// TwinCAT 3 PLC project Untitled1
// Title: Lib
// Company: Terza-Automation
// ProjectVersion: 0.1
// ProgramVersion: 3.1.4024.0
// libraries:
//   Tc2_ModbusRTU, * (Beckhoff Automation GmbH)
//   Tc2_Standard, * (Beckhoff Automation GmbH)
//   Tc2_System, * (Beckhoff Automation GmbH)
//   Tc2_Utilities, * (Beckhoff Automation GmbH)
//   Tc3_Module, * (Beckhoff Automation GmbH)
// project tree:
//   DUTs/ Beckhoff_AI.TcDUT, ModbusRealWordUnion.TcDUT, RTU_EM.TcDUT, RTU_STS.TcDUT, RTU_THT.TcDUT
//   / GlobalTextList.TcGTLO, PlcTask.TcTTO
//   GVLs/ GVL.TcGVL, GVL_DataHalls.TcGVL, GVL_DECI.TcGVL, GVL_Electrical.TcGVL, GVL_EM.TcGVL, GVL_STS.TcGVL, GVL_THT.TcGVL
//   POUs/ AccumDDHHMM.TcPOU, AccumTimes.TcPOU, CAC_Analog.TcPOU, CAC_Average.TcPOU, CAC_Mirror.TcPOU, MAIN.TcPOU, ModbusRTU_STS.TcPOU, ModbusRTU_THT.TcPOU, Modbus_EM.TcPOU, OneATS.TcPOU, OneCRAH.TcPOU, OneDI.TcPOU, OneEnergyMeter.TcPOU, OneFire_Suppr.TcPOU, OneGen.TcPOU, OneIDF.TcPOU, OneMYAUX_GLP.TcPOU, OnePDU.TcPOU, OneSTS.TcPOU, OneSWBL.TcPOU, OneTie_BRK.TcPOU, OneUPS.TcPOU
//   Version/ Global_Version.TcGVL
// real-time tasks:
//   TASK PlcTask: cycle T#10ms, priority 20, ADS port 350

CONFIGURATION Untitled1
    RESOURCE PLC ON TwinCAT3
        TASK PlcTask(INTERVAL := T#10ms, PRIORITY := 20);
        PROGRAM MAIN WITH PlcTask : MAIN;
    END_RESOURCE
END_CONFIGURATION

// ---- DUTs/Beckhoff_AI.TcDUT
TYPE Beckhoff_AI :
STRUCT
	rawValue : WORD;
	OutOfRange : BOOL;
	Offline : BOOL;
	Value : REAL;
	
END_STRUCT
END_TYPE

// ---- DUTs/ModbusRealWordUnion.TcDUT
TYPE ModbusRealWordUnion :
UNION
	realValue : REAL;
	wordValue : ARRAY[1..2] OF WORD;
END_UNION
END_TYPE

// ---- DUTs/RTU_EM.TcDUT
TYPE RTU_EM :
STRUCT
	Status : WORD;
	Operating_Hrs : REAL;
	Energy : REAL;
	Volume : REAL;
	Supply_Temp : REAL;
	Return_Temp : REAL;
	Temp_Diff : REAL;
	CommsError : BOOL;
	CommsErrorCode : INT;
END_STRUCT
END_TYPE

// ---- DUTs/RTU_STS.TcDUT
TYPE RTU_STS :
STRUCT
	CommsError : BOOL;
	CommsErrorCode : INT;

	PRI_VA : REAL;
	PRI_VB : REAL;
	PRI_VC : REAL;
	OTP_VA : REAL;
	OTP_VB : REAL;
	OTP_VC : REAL;
	AMPSA : REAL;
	AMPSB : REAL;
	AMPSC : REAL;
	FREQ : REAL;
	SEC_VA : REAL;
	SEC_VB : REAL;
	SEC_VC : REAL;
	OTP_LOAD_A : REAL;
	OTP_LOAD_B : REAL;
	OTP_LOAD_C : REAL;
	COM_ALM : BOOL;
	OTP_KW_A : REAL;
	OTP_KW_B : REAL;
	OTP_KW_C : REAL;
	OTP_KVA_A : REAL;
	OTP_KVA_B : REAL;
	OTP_KVA_C : REAL;
	PF_A : REAL;
	PF_B : REAL;
	PF_C : REAL;

	OTP_BKR_OPN : BOOL;
	L1_INP_BKR_OPN : BOOL;
	L2_INP_BKR_OPN : BOOL;
	L1_BYP_BKR_TRP : BOOL;
	L2_BYP_BKR_TRP : BOOL;
	OTP_BKR_TRP : BOOL;
	L1_INP_BKR_TRP : BOOL;
	L2_INP_BKR_TRP : BOOL;
	FANS_FAIL : BOOL;
	
END_STRUCT
END_TYPE

// ---- DUTs/RTU_THT.TcDUT
TYPE RTU_THT :
STRUCT
	Temp : REAL;
	RH : REAL;
	Temp_OOR : BOOL;
	RH_OOR : BOOL;
	CommsError : BOOL;
	CommsErrorCode : INT;
END_STRUCT
END_TYPE

// ---- GVLs/GVL.TcGVL
	{attribute 'qualified_only'}
VAR_GLOBAL
	mb_Input_Coils    	:	ARRAY [0..511] OF BOOL;
	mb_Output_Coils 	:   ARRAY [0..511] OF BOOL;
 	mb_Input_Registers 	:   ARRAY [0..511] OF WORD;
 	mb_Output_Registers :   ARRAY [0..255] OF WORD;
	
	nInputCoilIndex: INT;
	nOutputCoilIndex: INT;
	nInputRegisterIndex: INT;
	nOutputRegisterIndex: INT;
END_VAR

// ---- GVLs/GVL_DataHalls.TcGVL
{attribute 'qualified_only'}

VAR_GLOBAL CONSTANT
	StartInputCoilIndex_CRAH : INT := 0;			// uses 0-95
	StartInputCoilIndex_PDU : INT := 96;			// uses 96-239
	StartInputCoilIndex_CAC : INT := 0;				// not used
	StartInputCoilIndex_OtherDIs : INT := 275;		// uses 275-294
	StartInputCoilIndex_E_METER : INT := 295;		// uses 295-296
	StartInputCoilIndex_IO : INT := 297;			// uses 297-336
	StartInputCoilIndex_IDF : INT := 240;           // uses 240-257
	StartInputCoilIndex_GLP : INT := 258;           // uses 258-266
	StartInputCoilIndex_ATS : INT := 267;           // uses 267-274
    
	StartOutputCoilIndex_CRAH : INT := 0;			// uses 0-31
	StartOutputCoilIndex_PDU : INT := 0;			// not used
	StartOutputCoilIndex_CAC : INT := 35;			// uses 35-402
	StartOutputCoilIndex_OtherDIs : INT := 0;		// not used
	StartoutputCoilIndex_E_METER : INT := 0;		// not used
	StartoutputCoilIndex_IO : INT := 0;				// not used
	StartoutputCoilIndex_IDF : INT := 0;	        // not used
	StartoutputCoilIndex_GLP : INT := 0;	        // not used
	StartoutputCoilIndex_ATS : INT := 32;	        // uses 32-34
	
	StartInputRegisterIndex_CRAH: INT := 0;			// uses 0-127
	StartInputRegisterIndex_PDU: INT := 0;			// not used
	StartInputRegisterIndex_CAC: INT := 0;			// not used
	StartInputRegisterIndex_OtherDIs : INT := 0;	// not used
	StartInputRegisterIndex_E_METER : INT := 128;	// uses 128-254
    StartInputRegisterIndex_IO : INT := 0;			// not used
	StartInputRegisterIndex_IDF : INT := 0;			// not used
	StartInputRegisterIndex_GLP : INT := 0;			// not used
	StartInputRegisterIndex_ATS : INT := 0;			// not used
		
	StartOutputRegisterIndex_CRAH: INT := 0;		// not used
	StartOutputRegisterIndex_PDU: INT := 0;			// not used
	StartOutputRegisterIndex_CAC: INT := 0;			// uses 0-143
	StartOutputRegisterIndex_OtherDIs : INT := 0;	// not used
	StartoutputRegisterIndex_E_METER : INT := 0;	// not used
	StartoutputRegisterIndex_IO : INT := 0;			// not used
	StartoutputRegisterIndex_IDF : INT := 0;		// not used
	StartoutputRegisterIndex_GLP : INT := 0;		// not used
	StartoutputRegisterIndex_ATS : INT := 0;		// not used
	
END_VAR

// ---- GVLs/GVL_DECI.TcGVL
{attribute 'qualified_only'}
VAR_GLOBAL
	//Date and Time
    fbGetLocalSystemTime: FB_LocalSystemTime;
	sSystemDateTime : STRING;
	sSystemTime : STRING;
	sSystemDate : STRING;	

	// Coupler state - a UINT that should be 8 if its healthy
	CouplerStatus AT %I* : UINT;
	Term02Status AT %I* : WORD;
	Term03Status AT %I* : WORD;
	Term04Status AT %I* : WORD;
	Term05Status AT %I* : WORD;
	Term06Status AT %I* : WORD;
	Term07Status AT %I* : WORD;
	Term08Status AT %I* : WORD;
	Term09Status AT %I* : WORD;
	Term10Status AT %I* : WORD;
	Term11Status AT %I* : WORD;
	Term12Status AT %I* : WORD;
	Term13Status AT %I* : WORD;
	Term14Status AT %I* : WORD;
	Term15Status AT %I* : WORD;
	Term16Status AT %I* : WORD;
	Term17Status AT %I* : WORD;
	Term18Status AT %I* : WORD;
	Term19Status AT %I* : WORD;
	Term20Status AT %I* : WORD;
	Term21Status AT %I* : WORD;
	Term22Status AT %I* : WORD;
	Term23Status AT %I* : WORD;
	Term24Status AT %I* : WORD;
	Term25Status AT %I* : WORD;
	Term26Status AT %I* : WORD;
	Term27Status AT %I* : WORD;
	Term28Status AT %I* : WORD;
	Term29Status AT %I* : WORD;
	Term30Status AT %I* : WORD;
	Term31Status AT %I* : WORD;
	Term32Status AT %I* : WORD;
	Term33Status AT %I* : WORD;
	Term34Status AT %I* : WORD;
	Term35Status AT %I* : WORD;
	Term36Status AT %I* : WORD;
    Term37Status AT %I* : WORD;
	
	// I/O module status
	CouplerOffline : BOOL;
	Term02Offline : BOOL;
	Term03Offline : BOOL;
	Term04Offline : BOOL;
	Term05Offline : BOOL;
	Term06Offline : BOOL;
	Term07Offline : BOOL;
	Term08Offline : BOOL;
	Term09Offline : BOOL;
	Term10Offline : BOOL;
	Term11Offline : BOOL;
	Term12Offline : BOOL;
	Term13Offline : BOOL;
	Term14Offline : BOOL;
	Term15Offline : BOOL;
	Term16Offline : BOOL;
	Term17Offline : BOOL;
	Term18Offline : BOOL;
	Term19Offline : BOOL;
	Term20Offline : BOOL;
	Term21Offline : BOOL;
	Term22Offline : BOOL;
	Term23Offline : BOOL;
	Term24Offline : BOOL;
	Term25Offline : BOOL;
	Term26Offline : BOOL;
	Term27Offline : BOOL;
	Term28Offline : BOOL;
	Term29Offline : BOOL;
	Term30Offline : BOOL;
	Term31Offline : BOOL;
	Term32Offline : BOOL;
	Term33Offline : BOOL;
	Term34Offline : BOOL;
	Term35Offline : BOOL;
	Term36Offline : BOOL;
	Term37Offline : BOOL;
	
END_VAR

VAR_GLOBAL CONSTANT
	

END_VAR

// ---- GVLs/GVL_Electrical.TcGVL
{attribute 'qualified_only'}


VAR_GLOBAL CONSTANT
	StartInputCoilIndex_CRAH : INT := 0;			     // uses 0-29
	StartInputCoilIndex_SWBL : INT := 30;			     // uses 30-89
	StartInputCoilIndex_CAC : INT := 0;				     // not used
	StartInputCoilIndex_OtherDIs : INT := 297;		     // uses 297-330
	StartInputCoilIndex_TX : INT := 227;			     // uses 227-234
	StartInputCoilIndex_GEN : INT := 235;			     // uses 235-244
	StartInputCoilIndex_UPS : INT := 245;			     // uses 245-260
	StartInputCoilIndex_EMG_LIT : INT := 261;			 // uses 261-272
	StartInputCoilIndex_Fire_Suppr : INT := 273;		 // uses 273-296
	StartInputCoilIndex_ATS : INT := 219;                // uses 219-226
	StartInputCoilIndex_MYAUX_GLP : INT := 210;          // uses 210-218
	StartInputCoilIndex_Tie_BRK : INT := 90;             // uses 90-97
	StartInputCoilIndex_STS : INT := 98;			     // uses 98-209
	StartInputCoilIndex_STSRTU : INT := 331;		     // uses 331-407
 	StartInputCoilIndex_IO : INT := 408;				 // uses 408-430
 	StartInputCoilIndex_RTUStat : INT := 431;		 	 // uses 431-440
   
	StartOutputCoilIndex_CRAH : INT := 0;			     // uses 0-11
	StartOutputCoilIndex_SWBL : INT := 0;			     // not used
	StartOutputCoilIndex_CAC : INT := 23;			     // uses 23-52
	StartOutputCoilIndex_OtherDIs : INT := 0;		     // not used 
	StartOutputCoilIndex_TX : INT := 0;				     // not used
	StartOutputCoilIndex_GEN : INT := 53;	             // uses 53-54
	StartOutputCoilIndex_UPS : INT := 0;	             // not used
	StartOutputCoilIndex_EMG_LIT : INT := 0;	         // not used 
	StartOutputCoilIndex_Fire_Suppr : INT := 0;	         // not used
	StartOutputCoilIndex_ATS : INT := 20;	             // uses 20-22
	StartOutputCoilIndex_MYAUX_GLP : INT := 0;	         // not used
	StartOutputCoilIndex_Tie_BRK : INT := 0;	         // not used
	StartOutputCoilIndex_STS : INT := 12;	             // uses 12-19
	StartOutputCoilIndex_STSRTU : INT := 0;	             // not used
 	StartOutputCoilIndex_IO : INT := 0;				 	 // not used
 	StartOutputCoilIndex_RTUStat : INT := 0;			 // not used
	
	StartInputRegisterIndex_CRAH: INT := 0;			     // uses 0-46
	StartInputRegisterIndex_SWBL: INT := 0;			     // not used
	StartInputRegisterIndex_CAC: INT := 0;			     // not used
	StartInputRegisterIndex_OtherDIs : INT := 0;	     // not used
    StartInputRegisterIndex_TX : INT := 0;			     // not used
	StartInputRegisterIndex_GEN : INT := 0;			     // not used
	StartInputRegisterIndex_UPS : INT := 0;			     // not used
	StartInputRegisterIndex_EMG_LIT : INT := 0;			 // not used
	StartInputRegisterIndex_Fire_Suppr : INT := 0;	     // not used
	StartInputRegisterIndex_ATS : INT := 0;			     // not used
	StartInputRegisterIndex_MYAUX_GLP : INT := 0;	     // not used
	StartInputRegisterIndex_Tie_BRK : INT := 0;	         // not used
	StartInputRegisterIndex_STS : INT := 0;			     // not used
	StartInputRegisterIndex_STSRTU : INT := 61;			 // uses 61-460
 	StartInputRegisterIndex_IO : INT := 0;				 // not used
 	StartInputRegisterIndex_RTUStat : INT := 47;		 // uses 47-56
		
	StartOutputRegisterIndex_CRAH: INT := 0;		     // not used
	StartOutputRegisterIndex_SWBL: INT := 0;		     // not used
	StartOutputRegisterIndex_CAC: INT := 0;			     // uses 0-10
	StartOutputRegisterIndex_OtherDIs : INT := 0;	     // not used
	StartOutputRegisterIndex_TX : INT := 0;			     // not used
	StartOutputRegisterIndex_GEN : INT := 0;			 // not used
	StartOutputRegisterIndex_UPS : INT := 0;			 // not used
	StartOutputRegisterIndex_EMG_LIT : INT := 0;	     // not used
	StartOutputRegisterIndex_Fire_Suppr : INT := 0;	     // not used
	StartOutputRegisterIndex_ATS : INT := 0;		     // not used
	StartOutputRegisterIndex_MYAUX_GLP : INT := 0;		 // not used
	StartOutputRegisterIndex_Tie_BRK : INT := 0;		 // not used
	StartOutputRegisterIndex_STS : INT := 0;			 // not used
	StartOutputRegisterIndex_STSRTU : INT := 0;			 // not used
 	StartOutputRegisterIndex_IO : INT := 0;				 // not used
 	StartOutputRegisterIndex_RTUStat : INT := 0;		 // not used
	
END_VAR

// ---- GVLs/GVL_EM.TcGVL
{attribute 'qualified_only'}
VAR_GLOBAL
	EM : ARRAY [1..2] OF RTU_EM;
END_VAR

// ---- GVLs/GVL_STS.TcGVL
{attribute 'qualified_only'}
VAR_GLOBAL
	STS : ARRAY [1..10] OF RTU_STS;
END_VAR

// ---- GVLs/GVL_THT.TcGVL
{attribute 'qualified_only'}
VAR_GLOBAL
	THT : ARRAY [1..14] OF RTU_THT;
END_VAR


VAR_GLOBAL CONSTANT
	Temp_OOR_Min : REAL :=   0.0;
	Temp_OOR_Max : REAL :=  50.0;
	RH_OOR_Min   : REAL :=   0.0;
	RH_OOR_Max   : REAL := 100.0;
END_VAR

// ---- Version/Global_Version.TcGVL
{attribute 'TcGenerated'}
{attribute 'no-analysis'}
{attribute 'linkalways'}
// This function has been automatically generated from the project information.
VAR_GLOBAL CONSTANT
	{attribute 'const_non_replaced'}
	stLibVersion_Lib : ST_LibVersion := (iMajor := 0, iMinor := 1, iBuild := 0, iRevision := 0, nFlags := 0, sVersion := '0.1');
END_VAR

// ---- POUs/MAIN.TcPOU
PROGRAM MAIN
VAR
	foo:AccumDDHHMM;
	in1 AT %I* : BOOL;
	
	foo1: BOOL;
	foo2: BOOL;
	foo3: BOOL;
	
	foo4:STRING;
	
END_VAR

foo(State:=foo1 , Retentive:= foo2, Reset:=foo3);

foo4:=foo.DispayTime;

END_PROGRAM

// ---- POUs/AccumDDHHMM.TcPOU
FUNCTION_BLOCK AccumDDHHMM
VAR_INPUT
	State:BOOL;
	Retentive:BOOL;
	Reset:BOOL;
END_VAR

VAR PERSISTENT
	Mins:WORD;
	Hrs:WORD;
	Sec:WORD;
	Days:WORD;
END_VAR

VAR
	DispayTime:STRING;
	timer:TON;
	timerPT:TIME:=T#1M;
	StateToOff: F_TRIG;
    
END_VAR

VAR_TEMP
	displayTimeFormat: FB_FormatString;	
	foo:DINT;
END_VAR
VAR // added by the converter: edge detectors and wires of the graphical bodies
    _w1, _w2, _w3 : BOOL;
END_VAR

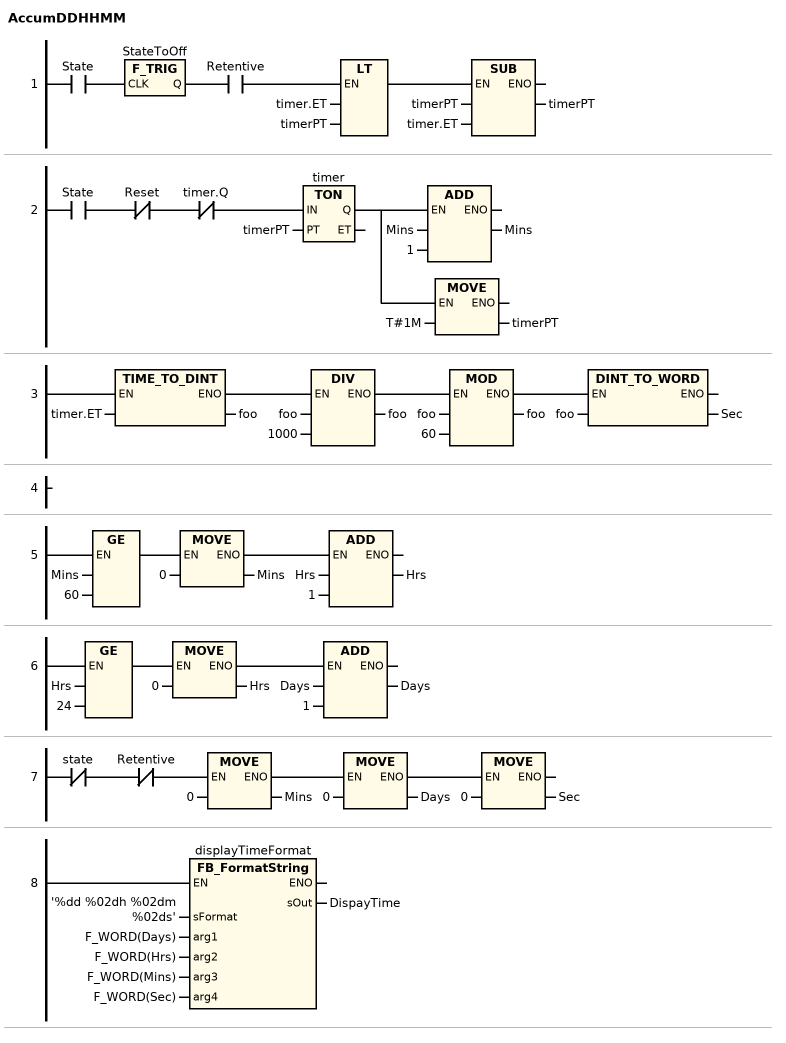
// NETWORK 1
StateToOff(CLK := State); // F_TRIG
IF StateToOff.Q AND Retentive AND timer.ET < timerPT THEN timerPT := timerPT - timer.ET; END_IF

// NETWORK 2
timer(IN := State AND NOT Reset AND NOT timer.Q, PT := timerPT); // TON
IF timer.Q THEN Mins := Mins + 1; END_IF
IF timer.Q THEN timerPT := T#1M; END_IF

// NETWORK 3
foo := TIME_TO_DINT(timer.ET);
foo := foo / 1000;
foo := foo MOD 60;
Sec := DINT_TO_WORD(foo);

// NETWORK 4

// NETWORK 5
_w1 := Mins >= 60;
IF _w1 THEN Mins := 0; END_IF
IF _w1 THEN Hrs := Hrs + 1; END_IF

// NETWORK 6
_w2 := Hrs >= 24;
IF _w2 THEN Hrs := 0; END_IF
IF _w2 THEN Days := Days + 1; END_IF

// NETWORK 7
_w3 := NOT state AND NOT Retentive;
IF _w3 THEN Mins := 0; END_IF
IF _w3 THEN Days := 0; END_IF
IF _w3 THEN Sec := 0; END_IF

// NETWORK 8
displayTimeFormat(
    sFormat := '%dd %02dh %02dm %02ds',
    arg1 := F_WORD(Days),
    arg2 := F_WORD(Hrs),
    arg3 := F_WORD(Mins),
    arg4 := F_WORD(Sec),
    sOut => DispayTime); // FB_FormatString

END_FUNCTION_BLOCK

// ---- POUs/AccumTimes.TcPOU
FUNCTION_BLOCK AccumTimes
VAR_INPUT
	State:BOOL;
END_VAR
VAR PERSISTENT
	Num:WORD;
	ResetAccum:BOOL;
	
	cntOn:CTU;
	Accum:AccumDDHHMM;
	On:AccumDDHHMM;
	Off:AccumDDHHMM;
END_VAR

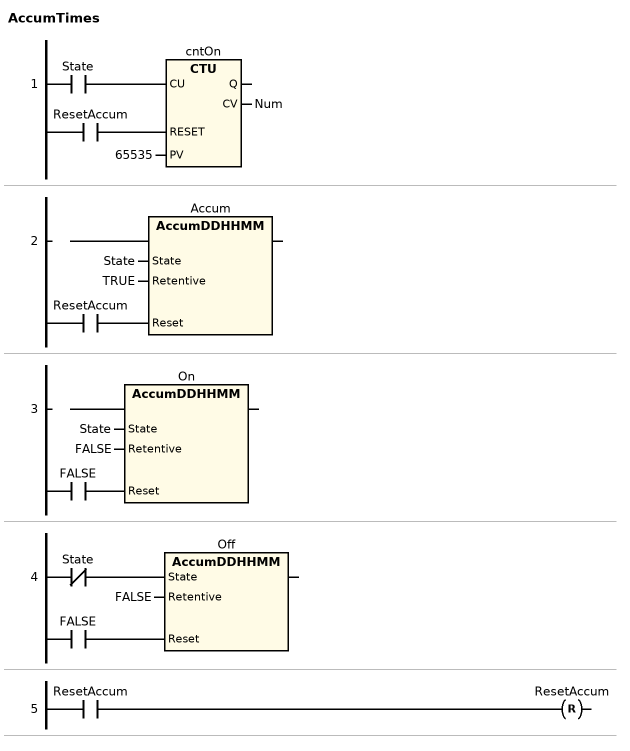
// NETWORK 1
cntOn(CU := State, RESET := ResetAccum, PV := 65535, CV => Num); // CTU

// NETWORK 2
Accum(State := State, Retentive := TRUE, Reset := ResetAccum); // AccumDDHHMM

// NETWORK 3
On(State := State, Retentive := FALSE, Reset := FALSE); // AccumDDHHMM

// NETWORK 4
Off(State := NOT State, Retentive := FALSE, Reset := FALSE); // AccumDDHHMM

// NETWORK 5
ResetAccum R= ResetAccum;

END_FUNCTION_BLOCK

// ---- POUs/CAC_Analog.TcPOU
FUNCTION_BLOCK CAC_Analog
VAR_INPUT
	Value : REAL;			// from EtherCAT I/O
	OutOfRange : BOOL;		// from EtherCAT I/O
	Offline: BOOL;			// from EtherCAT I/O
END_VAR

VAR
	SetInclude : BOOL;		// set on graphics, reset by WinCC OA
	SetExclude : BOOL;		// set on graphics, reset by WinCC OA
	Excluded : BOOL;		// maintained by WinCC OA
	Alarm : BOOL;			// maintained by WinCC OA
	SetIncludeTrig: R_TRIG;	
	SetExcludeTrig: R_TRIG;
END_VAR
VAR_TEMP
	i: INT;	
	modbusReal : ModbusRealWordUnion;
END_VAR


i := GVL.nOutputRegisterIndex;
modbusReal.realValue :=Value;
GVL.mb_Output_Registers[i+0]:= modbusReal.wordValue[1];
GVL.mb_Output_Registers[i+1]:= modbusReal.wordValue[2];

i := GVL.nOutputCoilIndex;
GVL.mb_Output_Coils[i+0]:=OutOfRange;
GVL.mb_Output_Coils[i+1]:=Offline;

SetIncludeTRig(CLK:=SetInclude);

IF SetIncludeTRig.Q THEN
	GVL.mb_Output_Coils[i+2]:=TRUE;
ELSIF SetInclude AND GVL.mb_Output_Coils[i+2] =0 THEN 
	SetInclude:= FALSE;
END_IF

END_FUNCTION_BLOCK

// ---- POUs/CAC_Average.TcPOU
FUNCTION_BLOCK CAC_Average
VAR_INPUT
END_VAR
VAR_OUTPUT
END_VAR
VAR
	Value:REAL;
	Alarm: BOOL;
	OutOfRange: BOOL;
	Offline: BOOL;
	
END_VAR

VAR_TEMP
	i : INT;
	modbusReal : ModbusRealWordUnion;
END_VAR


i:=GVL.nOutputRegisterIndex;
modbusReal.wordValue[0]:=GVL.mb_Output_Registers[i+0];
modbusReal.wordValue[1]:=GVL.mb_Output_Registers[i+1];
Value:= modbusReal.realValue;
GVL.nOutputRegisterIndex:=i+2;

i:=GVL.nOutputCoilIndex;
OutOfRange:=FALSE;
Offline:=GVL.mb_Output_Coils[i+0];
Alarm:=GVL.mb_Output_Coils[i+1];
GVL.nOutputCoilIndex:=i+2;

END_FUNCTION_BLOCK

// ---- POUs/CAC_Mirror.TcPOU
FUNCTION_BLOCK CAC_Mirror
VAR_INPUT
END_VAR
VAR_OUTPUT
END_VAR
VAR
	Value : REAL;			// from partner's EtherCAT I/O, via WinCC OA
	OutOfRange : BOOL;		// from partner's EtherCAT I/O, via WinCC OA
	Offline: BOOL;			// from partner's EtherCAT I/O, via WinCC OA
	SetInclude : BOOL;		// set on graphics, reset by WinCC OA
	SetExclude : BOOL;		// set on graphics, reset by WinCC OA
	Excluded : BOOL;		// maintained by WinCC OA
	Alarm : BOOL;			// maintained by WinCC OA
	SetIncludeTrig: R_TRIG;	
	SetExcludeTrig: R_TRIG;
END_VAR

VAR_TEMP
	i: INT;	
	modbusReal : ModbusRealWordUnion;
END_VAR


i := GVL.nOutputRegisterIndex;
modbusReal.wordValue[1] := GVL.mb_Output_Registers[i+0];
modbusReal.wordValue[2] := GVL.mb_Output_Registers[i+1];
Value := modbusReal.realValue;
GVL.nOutputRegisterIndex := i+2;


i := GVL.nOutputCoilIndex;
OutOfRange := GVL.mb_Output_Coils[i+0];
Offline := GVL.mb_Output_Coils[i+1];

SetIncludeTrig(CLK:=SetInclude);
IF SetIncludeTrig.Q THEN
	GVL.mb_Output_Coils[i+2] := TRUE;
ELSIF SetInclude AND GVL.mb_Output_Coils[i+2] = 0 THEN
	SetInclude := FALSE;
END_IF

SetExcludeTrig(CLK:=SetExclude);
IF SetExcludeTrig.Q THEN
	GVL.mb_Output_Coils[i+3] := TRUE;
ELSIF SetExclude AND GVL.mb_Output_Coils[i+3] = 0 THEN
	SetExclude := FALSE;
END_IF

Excluded := GVL.mb_Output_Coils[i+4];
Alarm := GVL.mb_Output_Coils[i+5];
GVL.nOutputCoilIndex := i+6;

END_FUNCTION_BLOCK

// ---- POUs/ModbusRTU_STS.TcPOU
FUNCTION_BLOCK ModbusRTU_STS
VAR_INPUT
	MB_FirstUnitID: BYTE;
	MB_LastUnitID: BYTE;
END_VAR
VAR_OUTPUT
END_VAR
VAR
	ModbusTerm: ModbusRtuMaster_KL6x22B;
	
	MB_UnitID: BYTE:=0;
	MB_Address : WORD := 0;
	MB_Quantity : WORD := 2;
	MB_ReadData : ARRAY[1..15] OF WORD;
	
	MB_TrigRead : BOOL := FALSE;
	MB_CommState:(TRiGGER, TRIGGERED, WAIT_RESPONSE, SETUP_NEXT_MESSAGE) := TRIGGER;
	tmrDelay:TON;
	Execute: INT;
END_VAR

VAR	
	STSNum: INT;
	MessageNum: INT := 1;
END_VAR


VAR CONSTANT
	MAX_MESSAGE_NUM: INT:=1;
	MODBUS_DELAY: TIME:=T#0MS;
END_VAR

IF (MB_UnitID < MB_FirstUnitID) OR (MB_UnitID>MB_LastUnitID) THEN 
	MB_UnitID:=MB_FirstUnitID;
	STSNum:=1;
	MessageNum:=1;
	MB_Address:=1;
	MB_Quantity:=13;
END_IF


ModbusTerm.ReadRegs(
	UnitID:= MB_UnitID, 
	Quantity:= MB_Quantity, 
	MBAddr:= MB_Address-1, 
	cbLength:= SIZEOF(MB_ReadData), 
	pMemoryAddr:= ADR(MB_ReadData), 
	Execute:= MB_TrigRead, 
	Timeout:= T#100MS, 
	BUSY=> , 
	Error=> , 
	ErrorId=> , 
	cbRead=> );
	
	
CASE MB_CommState OF 
	TRiGGER:
		tmrDelay(IN:=TRUE, PT:=MODBUS_DELAY);
		IF tmrDelay.Q THEN 
			MB_TrigRead:=TRUE;
			MB_CommState:=TRIGGERED;		
		END_IF
		
	TRIGGERED:
			tmrDelay(IN:=FALSE, PT:=MODBUS_DELAY);
			MB_TrigRead:=FALSE;
			MB_CommState:=WAIT_RESPONSE;
			
	WAIT_RESPONSE:
			IF NOT ModbusTerm.BUSY THEN
				GVL_STS.STS[STSNum].CommsError:= ModbusTerm.Error;
				GVL_STS.STS[STSNum].CommsErrorCode:= ModbusTerm.ErrorId;
				
				IF NOT ModbusTerm.Error THEN 
					IF MessageNum = 1 THEN // extracts the values in 13 registers #1-13
						GVL_STS.STS[STSNum].PRI_VA := WORD_TO_REAL(MB_ReadData[1]);
						GVL_STS.STS[STSNum].PRI_VB := WORD_TO_REAL(MB_ReadData[2]);
						GVL_STS.STS[STSNum].PRI_VC := WORD_TO_REAL(MB_ReadData[3]);
						GVL_STS.STS[STSNum].PRI_VA := WORD_TO_REAL(MB_ReadData[4]);
						GVL_STS.STS[STSNum].OTP_VB := WORD_TO_REAL(MB_ReadData[5]);
						GVL_STS.STS[STSNum].OTP_VC := WORD_TO_REAL(MB_ReadData[6]);
						GVL_STS.STS[STSNum].AMPSA  := WORD_TO_REAL(MB_ReadData[7]);
						GVL_STS.STS[STSNum].AMPSB  := WORD_TO_REAL(MB_ReadData[8]);
						GVL_STS.STS[STSNum].AMPSC  := WORD_TO_REAL(MB_ReadData[9]);
						GVL_STS.STS[STSNum].FREQ   := WORD_TO_REAL(MB_ReadData[10]);
						GVL_STS.STS[STSNum].SEC_VA := WORD_TO_REAL(MB_ReadData[11]);
						GVL_STS.STS[STSNum].SEC_VB := WORD_TO_REAL(MB_ReadData[12]);
						GVL_STS.STS[STSNum].SEC_VC := WORD_TO_REAL(MB_ReadData[14]);

					 ELSIF MessageNum = 2 THEN // extracts the values in 3 registers #17-19
						GVL_STS.STS[STSNum].OTP_LOAD_A:=WORD_TO_REAL(MB_ReadData[1]);
						GVL_STS.STS[STSNum].OTP_LOAD_B:=WORD_TO_REAL(MB_ReadData[2]);
						GVL_STS.STS[STSNum].OTP_LOAD_C:=WORD_TO_REAL(MB_ReadData[3]);
						
					ELSIF MessageNum = 3 THEN 					
						// common alarm is bit 15 of register 41
						GVL_STS.STS[STSNum].COM_ALM :=MB_ReadData[1].15;
						// other alarms of interest are in register 43 
						GVL_STS.STS[STSNum].OTP_BKR_OPN    := MB_ReadData[3].0;
						GVL_STS.STS[STSNum].L1_INP_BKR_OPN := MB_ReadData[3].1;
						GVL_STS.STS[STSNum].L2_INP_BKR_OPN := MB_ReadData[3].2;
						GVL_STS.STS[STSNum].L1_BYP_BKR_TRP := MB_ReadData[3].3;
						GVL_STS.STS[STSNum].L2_BYP_BKR_TRP := MB_ReadData[3].4;
						GVL_STS.STS[STSNum].OTP_BKR_TRP    := MB_ReadData[3].5;
						GVL_STS.STS[STSNum].L1_INP_BKR_TRP := MB_ReadData[3].6;
						GVL_STS.STS[STSNum].L2_INP_BKR_TRP := MB_ReadData[3].7;
						GVL_STS.STS[STSNum].FANS_FAIL      := MB_ReadData[3].8;	
					
					ELSIF MessageNum = 4 THEN 
						GVL_STS.STS[STSNum].OTP_KW_A  := WORD_TO_REAL(MB_ReadData[1]) / 10.0;
						GVL_STS.STS[STSNum].OTP_KW_B  := WORD_TO_REAL(MB_ReadData[2]) / 10.0;
						GVL_STS.STS[STSNum].OTP_KW_C  := WORD_TO_REAL(MB_ReadData[3]) / 10.0;
						GVL_STS.STS[STSNum].OTP_KVA_A := WORD_TO_REAL(MB_ReadData[4]) / 10.0;
						GVL_STS.STS[STSNum].OTP_KVA_B := WORD_TO_REAL(MB_ReadData[5]) / 10.0;
						GVL_STS.STS[STSNum].OTP_KVA_C := WORD_TO_REAL(MB_ReadData[6]) / 10.0;
					
					ELSIF MessageNum = 5 THEN 
						GVL_STS.STS[STSNum].PF_A := WORD_TO_REAL(MB_ReadData[1]) / 100.0;
						GVL_STS.STS[STSNum].PF_B := WORD_TO_REAL(MB_ReadData[2]) / 100.0;
						GVL_STS.STS[STSNum].PF_C := WORD_TO_REAL(MB_ReadData[3]) / 100.0;	
			
					END_IF
				END_IF
				 
				MB_CommState:=SETUP_NEXT_MESSAGE;
		  END_IF;	 

	SETUP_NEXT_MESSAGE:
		MessageNum:=MessageNum+1;
		
		IF MessageNum > MAX_MESSAGE_NUM THEN 
			MessageNum:=1;
			MB_UnitID:=MB_UnitID+1;
			STSNum:=STSNum+1;	
		END_IF
		
		IF MessageNum = 1  THEN // extracts the values in 13 registers #1-13
			MB_Address:=1;
			MB_Quantity:=13;
			
		ELSIF MessageNum = 2 THEN  // extracts the values in 3 registers #17-19
			MB_Address:=17;
			MB_Quantity:=3;
			 
		ELSIF MessageNum = 3 THEN  // extracts the alarms - 4 registers #41-44
			MB_Address:=41;
			MB_Quantity:=4;
			
		ELSIF MessageNum = 4 THEN  // extracts the values in 6 registers #56-61
			MB_Address:=56;
			MB_Quantity:=6;
			
		ELSIF MessageNum = 5 THEN  // extracts the values in 3 registers #69-71
			MB_Address:=69;
			MB_Quantity:=3;
			
		END_IF 
		
		MB_CommState:=TRiGGER;	
	
END_CASE

END_FUNCTION_BLOCK

// ---- POUs/ModbusRTU_THT.TcPOU
FUNCTION_BLOCK ModbusRTU_THT
VAR_INPUT
	MB_FirstUnitID:BYTE;
	MB_LastUnitID:BYTE;
END_VAR
VAR_OUTPUT
END_VAR
VAR
	ModbusTerm: ModbusRtuMaster_KL6x22B;
	
	MB_UnitID: BYTE:=0;
	MB_Address: WORD:=25;
	MB_Quantity: WORD:=4;
	MB_ReadData: ARRAY[1..2] OF ModbusRealWordUnion;
	
	MB_TrigRead: BOOL:=FALSE;
	MB_CommState: (TRIGGER, TRIGGERED, WAIT_RESPONSE) := TRIGGER;
	tmrDelay: TON;
	

END_VAR

IF (MB_UnitID < MB_FirstUnitID) OR (MB_UnitID>MB_LastUnitID) THEN 
	MB_UnitID:=MB_FirstUnitID;
END_IF


ModbusTerm(
	UnitID:= MB_UnitID, 
	Quantity:= MB_Quantity, 
	MBAddr:= MB_Address, 
	cbLength:= SIZEOF(MB_ReadData), 
	pMemoryAddr:= ADR(MB_ReadData), 
	Execute:= MB_TrigRead, 
	Timeout:= T#2S, 
	BUSY=> , 
	Error=> , 
	ErrorId=> , 
	cbRead=> );
	
CASE MB_CommState OF 
	TRIGGER: 
		tmrDelay(IN:=TRUE, PT:=T#1S);
		IF tmrDelay.Q THEN 
			MB_TrigRead:=TRUE;
			MB_CommState:=TRIGGERED;
		END_IF
		
	TRIGGERED:
		tmrDelay(IN:=FALSE, PT:=T#1S);
		MB_TrigRead:=FALSE;
		MB_CommState:=WAIT_RESPONSE;
		
	WAIT_RESPONSE:
		IF NOT ModbusTerm.BUSY THEN
			GVL_THT.THT[MB_UnitID].CommsError:=ModbusTerm.Error;
			GVL_THT.THT[MB_UnitID].CommsErrorCode:=ModbusTerm.ErrorId;
			
			IF NOT ModbusTerm.Error THEN
				GVL_THT.THT[MB_UnitID].Temp:=MB_ReadData[1].realValue;
				GVL_THT.THT[MB_UnitID].RH  :=MB_ReadData[2].realValue;
				
				GVL_THT.THT[MB_UnitID].Temp_OOR:= (GVL_THT.THT[MB_UnitID].Temp < GVL_THT.Temp_OOR_Min) OR 
												  (GVL_THT.THT[MB_UnitID].Temp > GVL_THT.Temp_OOR_Max);
												  
				GVL_THT.THT[MB_UnitID].RH_OOR:= (GVL_THT.THT[MB_UnitID].RH < GVL_THT.RH_OOR_Min) OR 
												(GVL_THT.THT[MB_UnitID].RH > GVL_THT.RH_OOR_Max);
			END_IF
			
		MB_UnitID   := MB_UnitID+1;
		MB_CommState:= TRIGGER;
		END_IF
END_CASE

END_FUNCTION_BLOCK

// ---- POUs/Modbus_EM.TcPOU
FUNCTION_BLOCK Modbus_EM
VAR_INPUT
	MB_FirstUnitID: BYTE;
	MB_LastUnitID: BYTE;
END_VAR
VAR_OUTPUT
END_VAR
VAR
	ModbusTerm: ModbusRtuMaster_KL6x22B;
	
	MB_UnitID : BYTE := 0;
	MB_Address : WORD := 0;
	MB_Quantity : WORD := 2;
	MB_ReadData : ModbusRealWordUnion;

	MB_TrigRead : BOOL := FALSE;
	MB_CommState: (TRIGGER, TRIGGERED, WAIT_RESPONSE, SETUP_NEXT_MESSAGE) := TRIGGER;
	tmrDelay: TON;
END_VAR

VAR
	EMNum:INT;
	MessageNum:INT;
END_VAR

IF (MB_UnitID < MB_FirstUnitID) OR (MB_UnitID>MB_LastUnitID) THEN 
	
	MB_UnitID:=MB_FirstUnitID;
	EMNum:=1;
	MessageNum:=1;
	MB_Address:=0;

END_IF

ModbusTerm.ReadRegs(
	UnitID:= MB_UnitID, 
	Quantity:= MB_Quantity, 
	MBAddr:= MB_Address, 
	cbLength:= SIZEOF(MB_ReadData), 
	pMemoryAddr:= ADR(MB_ReadData), 
	Execute:= MB_TrigRead, 
	Timeout:= T#2S, 
	BUSY=> , 
	Error=> , 
	ErrorId=> , 
	cbRead=> );
	
CASE MB_CommState OF
	TRIGGER:
			tmrDelay(in:=TRUE, PT:=T#1S);
			
			IF tmrDelay.Q THEN 
				MB_TrigRead:=TRUE;
				MB_CommState:=TRIGGERED;
			END_IF
			
	TRIGGERED:
			tmrDelay(in:=FALSE, PT:=T#1S);
			MB_TrigRead:=FALSE;			
			MB_CommState:=WAIT_RESPONSE;

	WAIT_RESPONSE:
			
			IF NOT ModbusTerm.BUSY THEN 
				GVl_Em.EM[EMNum].CommsError:=ModbusTerm.Error;
				GVl_Em.EM[EMNum].CommsErrorCode:=ModbusTerm.ErrorId;
				
				IF NOT ModbusTerm.Error THEN
					IF MessageNum=1 THEN 
						GVl_Em.EM[EMNum].Status:= MB_ReadData.wordValue[2];
					ELSIF MessageNum=2 THEN 
						GVl_Em.EM[EMNum].Operating_Hrs:= MB_ReadData.realValue;
					ELSIF MessageNum=3 THEN 
						GVl_Em.EM[EMNum].Energy:= MB_ReadData.realValue;
					ELSIF MessageNum=4 THEN 
						GVl_Em.EM[EMNum].Volume:= MB_ReadData.realValue;
					ELSIF MessageNum=5 THEN
						GVl_Em.EM[EMNum].Supply_Temp:= MB_ReadData.realValue;
					ELSIF MessageNum=6 THEN
						GVl_Em.EM[EMNum].Return_Temp:= MB_ReadData.realValue;
					ELSIF MessageNum =7 THEN
						GVl_Em.EM[EMNum].Temp_Diff:= MB_ReadData.realValue;
					END_IF;	
				END_IF
				
				MB_CommState:=SETUP_NEXT_MESSAGE;
				
			END_IF
				
	SETUP_NEXT_MESSAGE:
			MessageNum:=MessageNum+1;
			
			IF MessageNum> 7 THEN 
				
				MessageNum:=1;
				MB_UnitID:=MB_UnitID+1;
				EMNum:=EMNum+1;
				
			END_IF

			IF MessageNum = 1    THEN
				MB_Address:=0; // read status in word 2
			ELSIF MessageNum = 2 THEN 
				MB_Address:=6; // read operating hours
			ELSIF MessageNum = 3 THEN 
				MB_Address:=100; // read energy
			ELSIF MessageNum = 4 THEN 
				MB_Address:=200; // read volume
			ELSIF MessageNum = 5 THEN 
				MB_Address:=800; // read supply temperature
			ELSIF MessageNum = 6 THEN
				MB_Address:=810; // read return temperature
			ELSIF MessageNum = 7 THEN 
				MB_Address:=820;
			END_IF
			
		MB_CommState :=TRIGGER;

END_CASE

END_FUNCTION_BLOCK

// ---- POUs/OneATS.TcPOU
FUNCTION_BLOCK OneATS
VAR_INPUT
	ATS_Avai: BOOL;
	ATS_Avai_Offline: BOOL;	
	ATS_SP1: BOOL;
	ATS_SP1_Offline:BOOL;
	ATS_SP2 : BOOL;
	ATS_SP2_Offline : BOOL;
	ATS_SP0 : BOOL;
	ATS_SP0_Offline : BOOL;
END_VAR

VAR_OUTPUT
	Net_Priority: BOOL;
	Source_Priority: BOOL;
	Inhibited: BOOL;

END_VAR

VAR_TEMP
	i :INT;
END_VAR


i:=GVL.nInputCoilIndex;

GVL.mb_Input_Coils[i+0] := ATS_Avai;
GVL.mb_Input_Coils[i+1] := ATS_Avai_Offline;

GVL.mb_Input_Coils[i+2] := ATS_SP1;
GVL.mb_Input_Coils[i+3] := ATS_SP1_Offline;

GVL.mb_Input_Coils[i+4] := ATS_SP2;
GVL.mb_Input_Coils[i+5] := ATS_SP2_Offline;

GVL.mb_Input_Coils[i+6] := ATS_SP0;
GVL.mb_Input_Coils[i+7] := ATS_SP0_Offline;

i:=GVL.nOutputCoilIndex;
Net_Priority:= GVL.mb_Output_Coils[i+0];
Source_Priority:= GVL.mb_Output_Coils[i+1];
Inhibited:= GVL.mb_Output_Coils[i+2];

GVL.nOutputCoilIndex:=i+3;

END_FUNCTION_BLOCK

// ---- POUs/OneCRAH.TcPOU
FUNCTION_BLOCK OneCRAH
VAR_INPUT
	Running:BOOL;
	Alarm	:BOOL;
	Iso1_1_Sts:BOOL;
	Iso1_2_Sts:BOOL;
	Offline:BOOL;
END_VAR
VAR_OUTPUT
	Enable:BOOL;
END_VAR

VAR PERSISTENT
	Maintenance:BOOL;
	Inhibited:BOOL;
	HOA:WORD;
	Run: AccumTimes;
	Alm: AccumTimes;
	Ena: AccumTimes;
	
END_VAR

VAR_TEMP
	i:INT;
	modbusReal: ModbusRealWordUnion;
END_VAR

Run(State:=Running);
Alm(State:=Alarm);
Ena(State:=Enable);


i:= GVl.nInputCoilIndex;
GVL.mb_Input_Coils[i+0]:= Running;
GVL.mb_Input_Coils[i+1]:= Alarm;
GVL.mb_Input_Coils[i+2]:= Offline;
GVL.mb_Input_Coils[i+3]:= Iso1_1_Sts;
GVL.mb_Input_Coils[i+4]:= Iso1_2_Sts;

GVl.nInputCoilIndex := i+5;

i:=GVL.nOutputCoilIndex;
Enable:= GVL.mb_Output_Coils[i+0];
Inhibited:= GVL.mb_Output_Coils[i+1];
GVL.nOutputCoilIndex:=i+2;


i:=GVL.nInputRegisterIndex;
GVL.mb_Input_Registers[i+0]:= HOA;
GVL.mb_Input_Registers[i+1]:= Run.num;

modbusReal.realValue:= WORD_TO_REAL(Run.Accum.Days) * 24.0 +
					   WORD_TO_REAL(Run.Accum.Hrs)  * 1.0  +
					   WORD_TO_REAL(Run.Accum.Mins) / 60.0;
					   
GVL.mb_Input_Registers[i+2]:= modbusReal.wordValue[1];
GVL.mb_Input_Registers[i+3]:= modbusReal.wordValue[2];

modbusReal.realValue:= WORD_TO_REAL(Run.On.Days) * 24.0 +
					   WORD_TO_REAL(Run.On.Days) * 1.0 +
					   WORD_TO_REAL(Run.On.Mins) / 60.0;
					   
					   
GVL.mb_Input_Registers[i+4]:= modbusReal.wordValue[1];
GVL.mb_Input_Registers[i+5]:= modbusReal.wordValue[2];					   
					   
					   
modbusReal.realValue:= WORD_TO_REAL(Run.Off.Days) * 24.0 +
					   WORD_TO_REAL(Run.Off.Days) * 1.0 +
					   WORD_TO_REAL(Run.Off.Mins) / 60.0;
					   
					   
GVL.mb_Input_Registers[i+6]:= modbusReal.wordValue[1];
GVL.mb_Input_Registers[i+7]:= modbusReal.wordValue[2];

GVL.nInputRegisterIndex:=i+8;

END_FUNCTION_BLOCK

// ---- POUs/OneDI.TcPOU
FUNCTION_BLOCK OneDI
VAR_INPUT
	
	Value  :BOOL;
	Offline:BOOL;
	
END_VAR

VAR_TEMP
	i: INT;
	
END_VAR


i :=GVL.nInputCoilIndex;

GVL.mb_Input_Coils[i+0]:=Value;
GVL.mb_Input_Coils[i+1]:=Offline;

GVL.nInputCoilIndex:= i+2;

END_FUNCTION_BLOCK

// ---- POUs/OneEnergyMeter.TcPOU
FUNCTION_BLOCK OneEnergyMeter
VAR_INPUT
	Status: WORD;
    Operating_Hrs: REAL;
	Energy : REAL;
    Volume: REAL; 
	Supply_Temp: REAL;
	Return_Temp: REAL;
	Temp_Diff: REAL;
	Offline: BOOL;
END_VAR
VAR_OUTPUT
END_VAR
VAR_TEMP
	i : INT;
	modbusReal : ModbusRealWordUnion;
END_VAR


i := GVL.nInputRegisterIndex;

GVL.mb_Input_Registers[i+0] := Status;

modbusReal.realValue := Operating_Hrs;
GVL.mb_Input_Registers[i+2] := modbusReal.wordValue[1];
GVL.mb_Input_Registers[i+3] := modbusReal.wordValue[2];

modbusReal.realValue := Energy;
GVL.mb_Input_Registers[i+4] := modbusReal.wordValue[1];
GVL.mb_Input_Registers[i+5] := modbusReal.wordValue[2];

modbusReal.realValue := Volume;
GVL.mb_Input_Registers[i+6] := modbusReal.wordValue[1];
GVL.mb_Input_Registers[i+7] := modbusReal.wordValue[2];

modbusReal.realValue := Supply_Temp;
GVL.mb_Input_Registers[i+8] := modbusReal.wordValue[1];
GVL.mb_Input_Registers[i+9] := modbusReal.wordValue[2];

modbusReal.realValue := Return_Temp;
GVL.mb_Input_Registers[i+10] := modbusReal.wordValue[1];
GVL.mb_Input_Registers[i+11] := modbusReal.wordValue[2];

modbusReal.realValue := Temp_Diff;
GVL.mb_Input_Registers[i+12] := modbusReal.wordValue[1];
GVL.mb_Input_Registers[i+13] := modbusReal.wordValue[2];

GVL.nInputRegisterIndex := i + 14;


i := GVL.nInputCoilIndex;

GVL.mb_Input_Coils[i+0] := Offline;

GVL.nInputcoilIndex := i + 1;

END_FUNCTION_BLOCK

// ---- POUs/OneFire_Suppr.TcPOU
FUNCTION_BLOCK OneFire_Suppr
VAR_INPUT
	Pnl_Alm : BOOL;
	Pnl_FLT : BOOL;
	Supp_Act : BOOL;
	Fire_Offline : BOOL;
END_VAR
VAR_OUTPUT
END_VAR
VAR_TEMP
	i : INT;
END_VAR


i := GVL.nInputCoilIndex;

GVL.mb_Input_Coils[i+0] := Pnl_Alm;
GVL.mb_Input_Coils[i+1] := Pnl_FLT;
GVL.mb_Input_Coils[i+2] := Supp_Act;
GVL.mb_Input_Coils[i+3] := Fire_Offline;

GVL.nInputCoilIndex := i + 4;

END_FUNCTION_BLOCK

// ---- POUs/OneGen.TcPOU
FUNCTION_BLOCK OneGen
VAR_INPUT
	 Value : BOOL;
	 Offline : BOOL;
END_VAR
VAR_OUTPUT
	  Gen_Oper_Mode : BOOL;
	  Gen_EMG_Shut : BOOL;
END_VAR
VAR_TEMP
	i: INT;
END_VAR

i := GVL.nInputCoilIndex;

GVL.mb_Input_Coils[i+0] := Value;
GVL.mb_Input_Coils[i+1] := Offline;

GVL.nInputCoilIndex := i + 2;

i := GVL.nOutputCoilIndex;

Gen_Oper_Mode := GVL.mb_Output_Coils[i+0];
Gen_EMG_Shut  := GVL.mb_Output_Coils[i+1];

GVL.nOutputCoilIndex := i+2;

END_FUNCTION_BLOCK

// ---- POUs/OneIDF.TcPOU
FUNCTION_BLOCK OneIDF
VAR_INPUT
	sur_STS :BOOL;
	phs_ALM :BOOL;
	sur_phs_offline :BOOL;
	
	BRK115_POS_STS  :BOOL;
	BRK115_TRIP_ALM :BOOL;
	BRK115_offline: BOOL;
	
    BRK125_POS_STS: BOOL;
	BRK125_TRIP_ALM : BOOL; 
	BRK125_offline: BOOL;
		
END_VAR
VAR_OUTPUT
END_VAR

VAR_TEMP
	
	i:INT;

END_VAR

i := GVL.nInputCoilIndex;

GVL.mb_Input_Coils[i+0]:= sur_STS;
GVL.mb_Input_Coils[i+1]:= phs_ALM; 
GVL.mb_Input_Coils[i+2]:= sur_phs_offline;

GVL.mb_Input_Coils[i+3]:= BRK115_POS_STS; 
GVL.mb_Input_Coils[i+4]:= BRK115_TRIP_ALM; 
GVL.mb_Input_Coils[i+5]:= BRK115_offline; 

GVL.mb_Input_Coils[i+6]:= BRK125_POS_STS; 
GVL.mb_Input_Coils[i+7]:= BRK125_TRIP_ALM; 
GVL.mb_Input_Coils[i+8]:= BRK125_offline;

GVL.nInputCoilIndex:=i+9;

END_FUNCTION_BLOCK

// ---- POUs/OneMYAUX_GLP.TcPOU
FUNCTION_BLOCK OneMYAUX_GLP
VAR_INPUT
	sur_STS : BOOL;
	phs_ALM : BOOL;
	sur_phs_offline : BOOL;
	
    BRK119_POS_STS: BOOL;
	BRK119_TRIP_ALM : BOOL; 
	BRK119_offline: BOOL;
	
    BRK129_POS_STS: BOOL;
	BRK129_TRIP_ALM : BOOL; 
	BRK129_offline: BOOL;
END_VAR
VAR_OUTPUT
END_VAR
VAR_TEMP
	i: INT;
END_VAR


i := GVL.nInputCoilIndex;

GVL.mb_Input_Coils[i+0] := sur_STS;
GVL.mb_Input_Coils[i+1] := phs_ALM;
GVL.mb_Input_Coils[i+2] := sur_phs_offline;

GVL.mb_Input_Coils[i+3] := BRK119_POS_STS;
GVL.mb_Input_Coils[i+4] := BRK119_TRIP_ALM;
GVL.mb_Input_Coils[i+5] := BRK119_offline;

GVL.mb_Input_Coils[i+6] := BRK129_POS_STS;
GVL.mb_Input_Coils[i+7] := BRK129_TRIP_ALM;
GVL.mb_Input_Coils[i+8] := BRK129_offline;

GVL.nInputCoilIndex := i + 9;

END_FUNCTION_BLOCK

// ---- POUs/OnePDU.TcPOU
FUNCTION_BLOCK OnePDU
VAR_INPUT
	sur_STS:BOOL;
	phs_ALM:BOOL;
	sur_phs_offline : BOOL;
	
	tvoc_BRK_STS: BOOL;             // CIRCUIT BREAERS
	tvoc_BRK_ALM: BOOL;            // CIRCUIT BREAERS
	tvoc_BRK_offline: BOOL; 
	
	BRK115_POS_STS: BOOL;
	BRK115_TRIP_ALM : BOOL; 
	BRK115_offline: BOOL;
	
	BRK125_POS_STS: BOOL;
	BRK125_TRIP_ALM : BOOL; 
	BRK125_offline: BOOL;
	
	BRK135_POS_STS: BOOL;
	BRK135_TRIP_ALM : BOOL; 
	BRK135_offline: BOOL;
	
	BRK215_POS_STS: BOOL;
	BRK215_TRIP_ALM : BOOL; 
	BRK215_offline: BOOL;
	
	BRK225_POS_STS: BOOL;
	BRK225_TRIP_ALM : BOOL; 
	BRK225_offline: BOOL;
	
	BRK235_POS_STS: BOOL;
	BRK235_TRIP_ALM : BOOL; 
	BRK235_offline: BOOL;
	
	BRK315_POS_STS: BOOL;
	BRK315_TRIP_ALM : BOOL; 
	BRK315_offline: BOOL;
	
	BRK325_POS_STS: BOOL;
	BRK325_TRIP_ALM : BOOL; 
	BRK325_offline: BOOL;
	
	BRK335_POS_STS: BOOL;
	BRK335_TRIP_ALM : BOOL; 
	BRK335_offline: BOOL;
	
	BRK345_POS_STS: BOOL;
	BRK345_TRIP_ALM : BOOL; 
	BRK345_offline: BOOL;
	
END_VAR

VAR_TEMP
	i: INT;
END_VAR


i := GVL.nInputCoilIndex;
GVL.mb_Input_Coils[i+0] := sur_STS;
GVL.mb_Input_Coils[i+1] := phs_ALM;
GVL.mb_Input_Coils[i+2] := sur_phs_offline;

GVL.mb_Input_Coils[i+3] := tvoc_BRK_STS ;
GVL.mb_Input_Coils[i+4] := tvoc_BRK_ALM ;
GVL.mb_Input_Coils[i+5] := tvoc_BRK_offline;

GVL.mb_Input_Coils[i+6] := BRK115_POS_STS;
GVL.mb_Input_Coils[i+7] := BRK115_TRIP_ALM;
GVL.mb_Input_Coils[i+8] := BRK115_offline;

GVL.mb_Input_Coils[i+9] := BRK125_POS_STS;
GVL.mb_Input_Coils[i+10] := BRK125_TRIP_ALM;
GVL.mb_Input_Coils[i+11] := BRK125_offline;

GVL.mb_Input_Coils[i+12] := BRK135_POS_STS;
GVL.mb_Input_Coils[i+13] := BRK135_TRIP_ALM;
GVL.mb_Input_Coils[i+14] := BRK135_offline;

GVL.mb_Input_Coils[i+15] := BRK215_POS_STS;
GVL.mb_Input_Coils[i+16] := BRK215_TRIP_ALM;
GVL.mb_Input_Coils[i+17] := BRK215_offline;

GVL.mb_Input_Coils[i+18] := BRK225_POS_STS;
GVL.mb_Input_Coils[i+19] := BRK225_TRIP_ALM;
GVL.mb_Input_Coils[i+20] := BRK225_offline;

GVL.mb_Input_Coils[i+21] := BRK235_POS_STS;
GVL.mb_Input_Coils[i+22] := BRK235_TRIP_ALM;
GVL.mb_Input_Coils[i+23] := BRK235_offline;

GVL.mb_Input_Coils[i+24] := BRK315_POS_STS;
GVL.mb_Input_Coils[i+25] := BRK315_TRIP_ALM;
GVL.mb_Input_Coils[i+26] := BRK315_offline;

GVL.mb_Input_Coils[i+27] := BRK325_POS_STS;
GVL.mb_Input_Coils[i+28] := BRK325_TRIP_ALM;
GVL.mb_Input_Coils[i+29] := BRK325_offline;

GVL.mb_Input_Coils[i+30] := BRK335_POS_STS;
GVL.mb_Input_Coils[i+31] := BRK335_TRIP_ALM;
GVL.mb_Input_Coils[i+32] := BRK335_Offline;

GVL.mb_Input_Coils[i+33] := BRK345_POS_STS;
GVL.mb_Input_Coils[i+34] := BRK345_TRIP_ALM;
GVL.mb_Input_Coils[i+35] := BRK345_Offline;

GVL.nInputCoilIndex := i + 36;

END_FUNCTION_BLOCK

// ---- POUs/OneSTS.TcPOU
FUNCTION_BLOCK OneSTS
VAR_INPUT
	
	Trans_Inhibt : BOOL;
	Trans_Inhibt_Offline : BOOL;
    Com_Alm : BOOL;
	Com_Alm_Offline: BOOL;
    Fan_Fail : BOOL;
	Fan_Fail_Offline : BOOL;
	
    Load_Line_1 : BOOL;
	Load_Line_1_Offline : BOOL;
    Load_Line_2 : BOOL;
	Load_Line_2_Offline : BOOL;
	
    Load_Line_1_ByPass : BOOL;
	LL_1_ByPass_offline : BOOL;
    Load_Line_2_ByPass : BOOL;
	LL_2_ByPass_offline : BOOL;
	Load_DisCon : BOOL;
	Load_DisCon_Offline : BOOL;

END_VAR
VAR_OUTPUT
	STS_Inhibited : BOOL;
END_VAR
VAR_TEMP
	i : INT;
END_VAR



i := GVL.nInputCoilIndex;
GVL.mb_Input_Coils[i+0] := Trans_Inhibt;
GVL.mb_Input_Coils[i+1] := Trans_Inhibt_Offline;

GVL.mb_Input_Coils[i+2] := Com_Alm;
GVL.mb_Input_Coils[i+3] := Com_Alm_Offline;

GVL.mb_Input_Coils[i+4] := Fan_Fail;
GVL.mb_Input_Coils[i+5] := Fan_Fail_Offline;

GVL.mb_Input_Coils[i+6] := Load_Line_1;
GVL.mb_Input_Coils[i+7] := Load_Line_1_Offline;

GVL.mb_Input_Coils[i+8] := Load_Line_2;
GVL.mb_Input_Coils[i+9] := Load_Line_2_Offline;

GVL.mb_Input_Coils[i+10] := Load_Line_1_ByPass;
GVL.mb_Input_Coils[i+11] := LL_1_ByPass_offline;

GVL.mb_Input_Coils[i+12] := Load_Line_2_ByPass;
GVL.mb_Input_Coils[i+13] := LL_2_ByPass_offline;

GVL.mb_Input_Coils[i+13] := Load_DisCon;
GVL.mb_Input_Coils[i+14] := Load_DisCon_Offline;

GVL.nInputCoilIndex := i + 15;


i := GVL.nOutputCoilIndex;
STS_Inhibited := GVL.mb_Output_Coils[i+0];
GVL.nOutputCoilIndex := i+1;

END_FUNCTION_BLOCK

// ---- POUs/OneSWBL.TcPOU
FUNCTION_BLOCK OneSWBL
VAR_INPUT
	sur_STS : BOOL;
	phs_ALM_1 : BOOL;
	phs_ALM_2 : BOOL;
	sur_phs_offline : BOOL;
	
	Etherm_24VDC_STS : BOOL;
	Etherm_24VDC_Offline: BOOL;
	
	tvoc_BRK_STS: BOOL;               // CIRCUIT BREAERS
	tvoc_BRK_ALM: BOOL; 
    tvoc_24VDC_STS : BOOL;           // CIRCUIT BREAERS
	tvoc_BRK_offline: BOOL; 
	
	BRK_FC11_POS_STS: BOOL;
	BRK_FC11_TRIP_ALM : BOOL; 
	BRK_FC11_offline: BOOL;
	
	BRK_BA01_POS_STS: BOOL;
	BRK_BA01_TRIP_ALM : BOOL; 
	BRK_BA01_offline: BOOL;
	
    BRK_EC01_POS_STS: BOOL;
	BRK_EC01_TRIP_ALM : BOOL; 
	BRK_EC01_offline: BOOL;
	
	BRK_JA01_POS_STS: BOOL;
	BRK_JA01_TRIP_ALM : BOOL; 
	BRK_JA01_offline: BOOL;
	
    BRK_MC01_POS_STS: BOOL;
	BRK_MC01_TRIP_ALM : BOOL; 
	BRK_MC01_offline: BOOL;
	
	BRK_RA01_POS_STS: BOOL;
	BRK_RA01_TRIP_ALM : BOOL; 
	BRK_RA01_offline: BOOL;
	
	
	BRK_NO2_BA01_POS_STS: BOOL;
	BRK_NO2_BA01_TRIP_ALM : BOOL; 
	BRK_NO2_BA01_offline: BOOL;
END_VAR
VAR_OUTPUT
END_VAR
VAR_TEMP
	i:INT;
END_VAR


i := GVL.nInputCoilIndex;
GVL.mb_Input_Coils[i+0] := sur_STS;
GVL.mb_Input_Coils[i+1] := phs_ALM_1;
GVL.mb_Input_Coils[i+2] := phs_ALM_2;
GVL.mb_Input_Coils[i+3] := sur_phs_offline;

GVL.mb_Input_Coils[i+4] := Etherm_24VDC_STS;
GVL.mb_Input_Coils[i+5] := Etherm_24VDC_Offline;

GVL.mb_Input_Coils[i+6] := tvoc_BRK_STS ;
GVL.mb_Input_Coils[i+7] := tvoc_BRK_ALM ;
GVL.mb_Input_Coils[i+8] := tvoc_24VDC_STS;
GVL.mb_Input_Coils[i+9] := tvoc_BRK_offline;

GVL.mb_Input_Coils[i+10] := BRK_FC11_POS_STS;
GVL.mb_Input_Coils[i+11] := BRK_FC11_TRIP_ALM;
GVL.mb_Input_Coils[i+12] := BRK_FC11_offline;

GVL.mb_Input_Coils[i+13] := BRK_BA01_POS_STS;
GVL.mb_Input_Coils[i+14] := BRK_BA01_TRIP_ALM;
GVL.mb_Input_Coils[i+15] := BRK_BA01_offline;

GVL.mb_Input_Coils[i+16] := BRK_EC01_POS_STS;
GVL.mb_Input_Coils[i+17] := BRK_EC01_TRIP_ALM;
GVL.mb_Input_Coils[i+18] := BRK_EC01_offline;

GVL.mb_Input_Coils[i+19] := BRK_JA01_POS_STS;
GVL.mb_Input_Coils[i+20] := BRK_JA01_TRIP_ALM;
GVL.mb_Input_Coils[i+21] := BRK_JA01_offline;

GVL.mb_Input_Coils[i+22] := BRK_MC01_POS_STS;
GVL.mb_Input_Coils[i+23] := BRK_MC01_TRIP_ALM;
GVL.mb_Input_Coils[i+24] := BRK_MC01_offline;

GVL.mb_Input_Coils[i+25] := BRK_RA01_POS_STS;
GVL.mb_Input_Coils[i+26] := BRK_RA01_TRIP_ALM;
GVL.mb_Input_Coils[i+27] := BRK_RA01_offline;

GVL.mb_Input_Coils[i+28] := BRK_NO2_BA01_POS_STS;
GVL.mb_Input_Coils[i+29] := BRK_NO2_BA01_TRIP_ALM;
GVL.mb_Input_Coils[i+30] := BRK_NO2_BA01_offline;

GVL.nInputCoilIndex := i + 31;

END_FUNCTION_BLOCK

// ---- POUs/OneTie_BRK.TcPOU
FUNCTION_BLOCK OneTie_BRK
VAR_INPUT
	
	TIEBKR_STS: BOOL;
	TIEBKR_STS_Offline: BOOL;
	
	TIEBKR_RCKIN : BOOL;
	TIEBKR_RCKIN_Offline : BOOL;
	
	TIEBKR_TEST : BOOL;
	TIEBKR_TEST_Offline : BOOL;
	
	TIEBKR_RCKOUT : BOOL;
	TIEBKR_RCKOUT_Offline : BOOL;
	
END_VAR
VAR_OUTPUT
END_VAR
VAR_TEMP
	i : INT;
END_VAR


i := GVL.nInputCoilIndex;

GVL.mb_Input_Coils[i+0] := TIEBKR_STS;
GVL.mb_Input_Coils[i+1] := TIEBKR_STS_Offline;

GVL.mb_Input_Coils[i+2] := TIEBKR_RCKIN;
GVL.mb_Input_Coils[i+3] := TIEBKR_RCKIN_Offline;

GVL.mb_Input_Coils[i+4] := TIEBKR_TEST;
GVL.mb_Input_Coils[i+5] := TIEBKR_TEST_Offline;

GVL.mb_Input_Coils[i+6] := TIEBKR_RCKOUT;
GVL.mb_Input_Coils[i+7] := TIEBKR_RCKOUT_Offline;

GVL.nInputCoilIndex := i + 8;

END_FUNCTION_BLOCK

// ---- POUs/OneUPS.TcPOU
FUNCTION_BLOCK OneUPS
VAR_INPUT
	Crit_Alm : BOOL;
	Minor_Alm : BOOL;
	ByPass_Mode : BOOL;
	Batt_Mode : BOOL;
	Offline : BOOL;
END_VAR
VAR_OUTPUT
END_VAR
VAR_TEMP
	 i : INT;
END_VAR

i := GVL.nInputCoilIndex;

GVL.mb_Input_Coils[i+0] := Crit_Alm;
GVL.mb_Input_Coils[i+1] := Minor_Alm;
GVL.mb_Input_Coils[i+2] := ByPass_Mode;
GVL.mb_Input_Coils[i+3] := Batt_Mode;
GVL.mb_Input_Coils[i+4] := Offline;

GVL.nInputCoilIndex := i + 5;

END_FUNCTION_BLOCK

// ---- GlobalTextList.TcGTLO
TEXTLIST GlobalTextList
  24 = '%s'
  714 = 'Accumulated Runtime'
  99 = 'asfd'
  334 = 'Close'
  120 = 'CRAH %s'
  389 = 'Disable Maintenance'
  216 = 'Enable Maintenance'
  734 = 'Number of Starts'
  148 = 'Operator Options'
  716 = 'Reset'
  46 = 'Running Timing'
  124 = 'Running Timings'
  646 = 'Set Auto'
  977 = 'Set Hand'
  766 = 'Set Off'
  898 = 'Time In Alarm'
  184 = 'Time Since Last Run'
END_TEXTLIST
